TYPE ST_RepeatHistory :
STRUCT
  bSelected       : BOOL;     // UI selected
  nIndex          : UDINT;    // list index
  nX0             : DINT;     // X0 detected position
  fLen            : LREAL;    // Length intended
  fLenEffective   : LREAL;    // Effective dist to previous
  fLenDiff        : LREAL;    // Length difference to image length
  bLenNotInRange  : BOOL;     // Effective length not in range
  bInvalidIngoredMarks : BOOL;// Invalid marks seen, but ignored
  bMissingMarks   : BOOL;     // Some missing marks seen
END_STRUCT
END_TYPE

(* stored: Version 1.1.0.1, ProductVersion 3.1.4024.11
   DUT ST_RepeatHistory: Id {94d14178-4632-42c6-ab3e-45022b89e73f} *)
